(*
SPDX-FileCopyrightText: © 2026 Oleksandr Tiutyk <trofimich@gmail.com>
SPDX-License-Identifier: MIT
License: https://opensource.org/license/mit
*)

(*!
<summary>
Beckhoff EL3002: 2-channel analog input terminal (-10 V .. +10 V, 12-bit).
</summary>
<description>
Process image mapping structure for the EL3002 EtherCAT terminal with 2 analog input channels.
When used for I/O, link located fields or their containing buffers to the matching selected PDOs.
The record is not a packed wire buffer; compiler padding is not part of the device specification.
Unlinked/default values do not prove valid I/O. The caller evaluates bus/channel validity before use.
Use one owner task per instance and externally synchronize other access; multi-field snapshots are not atomic.
Copies store data without creating hardware links. Keep borrowed field references valid while consumers are bound.
This passive record performs no validation, synchronization, configuration or protocol advancement.
Select standard status-plus-value PDOs matching the declared Value type; compact value-only PDOs
are outside this model. Configure electrical range and scaling separately on the device.
</description>
*)
TYPE EL3002 :
STRUCT
	Ch1 : ANALOG_INPUT_INT_CHANNEL;
	Ch2 : ANALOG_INPUT_INT_CHANNEL;
END_STRUCT
END_TYPE

(* stored: Version 1.1.0.1, ProductVersion 3.1.4026.20
   DUT EL3002: Id {2a48f6a9-f290-4be8-99a1-66d6f98e3c95} *)
